// TIA Portal V19 export
FUNCTION "MachineInterface_NotExist" : Void   // FC142, LAD
TITLE = MACHINE INYTREFACE CUMULTIVE
// stored: Access Published, SetENOAutomatically false
   VAR_OUTPUT
      MachineInterface : "MachineInterface";
   END_VAR
BEGIN

REGION Network 1 (SCL): Execute
   #MachineInterface.AutReady := TRUE;


   #MachineInterface.Aborting := FALSE;

   #MachineInterface.AckStopInPhase := TRUE;

   #MachineInterface.AckStopProgrammed := TRUE;

   #MachineInterface.MotionsStandStill := TRUE;

   #MachineInterface.AlarmsPresence := FALSE;


   #MachineInterface.WarningPresence := FALSE;
END_REGION
END_FUNCTION
